{attribute 'qualified_only'}
{attribute 'strict'}
TYPE E_SDSState :
(
    Standby,
    Error,
    Operating
) UINT;
END_TYPE

(* stored: Version 1.1.0.1
   DUT E_SDSState: Id {cfdcfd5d-528d-0a41-25de-36cc8f8caf6f} *)
